{attribute 'linkalways'} 
{attribute 'no_explicit_call' := 'This FB is a CLASS and must be accessed using methods or properties'}
{attribute 'enable_dynamic_creation'}
FUNCTION_BLOCK _ETcVnDiffusivityTypeKAZE EXTENDS EnumDatatypeBase
VAR
	localData : ETcVnDiffusivityTypeKAZE;
	activeData : REFERENCE TO ETcVnDiffusivityTypeKAZE;
	enumBaseDatatype : _DINT(localData);
END_VAR

METHOD PRIVATE AddLocalEnumeration
VAR_INPUT
	Enumeration : T_MAXSTRING;
	Value : ETcVnDiffusivityTypeKAZE;
END_VAR
AddEnumeration(Enumeration, Value);
END_METHOD

PROPERTY PUBLIC Address : PVOID
GET
Address := ADR(activeData);
END_GET
END_PROPERTY

METHOD PUBLIC ClearReference
VAR_INPUT
END_VAR
activeData REF= localData;
SetBaseDatatypeReference();
END_METHOD

METHOD PUBLIC Clone : I_Datatype
VAR
    pClone : POINTER TO _ETcVnDiffusivityTypeKAZE;
END_VAR
pClone := __NEW(_ETcVnDiffusivityTypeKAZE(InitialValue := Value));
Clone := pClone^;
END_METHOD

METHOD FB_init : BOOL
VAR_INPUT
	bInitRetains : BOOL; // if TRUE, the retain variables are initialized (warm start / cold start)
	bInCopyCode : BOOL;  // if TRUE, the instance afterwards gets moved into the copy code (online change)
	InitialValue : ETcVnDiffusivityTypeKAZE;
END_VAR
localData := InitialValue;
AddBaseDatatype(enumBaseDatatype);
ClearReference();

AddLocalEnumeration('TCVN_DT1_KAZE_PM_G1', ETcVnDiffusivityTypeKAZE.TCVN_DT1_KAZE_PM_G1);
AddLocalEnumeration('TCVN_DT1_KAZE_PM_G2', ETcVnDiffusivityTypeKAZE.TCVN_DT1_KAZE_PM_G2);
AddLocalEnumeration('TCVN_DT1_KAZE_WEICKERT', ETcVnDiffusivityTypeKAZE.TCVN_DT1_KAZE_WEICKERT);
AddLocalEnumeration('TCVN_DT1_KAZE_CHARBONNIER', ETcVnDiffusivityTypeKAZE.TCVN_DT1_KAZE_CHARBONNIER);
END_METHOD

PROPERTY PUBLIC Identifier : T_MAXSTRING
GET
Identifier := 'ETcVnDiffusivityTypeKAZE';
END_GET
END_PROPERTY

METHOD IsEnumeratorValueEqual : BOOL
VAR_INPUT
	Enumerator : I_KeyValueForwardEnumerator;
END_VAR
VAR
	storedValue : ETcVnDiffusivityTypeKAZE;
END_VAR
IF NOT Enumerator.TryGet(storedValue) THEN
	RETURN;
END_IF

IsEnumeratorValueEqual := storedValue = activeData;
END_METHOD

METHOD PUBLIC MakeReferenceTo
VAR_INPUT
	ReferenceTarget : REFERENCE TO ETcVnDiffusivityTypeKAZE;
END_VAR
activeData REF= ReferenceTarget;
SetBaseDatatypeReference();
END_METHOD

METHOD PROTECTED SetBaseDatatypeReference
VAR_INPUT
END_VAR
enumBaseDatatype.MakeReferenceTo(activeData);
END_METHOD

PROPERTY PUBLIC Size : UDINT
GET
Size := SIZEOF(activeData);
END_GET
END_PROPERTY

METHOD TryMakeReferenceTo : BOOL
VAR_INPUT
	Target : I_Datatype;
END_VAR
VAR
	pTargetData : POINTER TO ETcVnDiffusivityTypeKAZE;
END_VAR
IF NOT IsEquivalentTo(Target) THEN
	RETURN;
END_IF

pTargetData := Target.Address;
activeData REF= pTargetData^;
SetBaseDatatypeReference();
TryMakeReferenceTo := TRUE;
END_METHOD

PROPERTY PUBLIC Value : ETcVnDiffusivityTypeKAZE
GET
Value := activeData;
END_GET
SET
activeData := Value;
END_SET
END_PROPERTY

END_FUNCTION_BLOCK

(* stored: Version 1.1.0.1, ProductVersion 3.1.4024.13
   POU _ETcVnDiffusivityTypeKAZE: Id {44374c61-c9bd-0cab-393d-297717105bca}, SpecialFunc None
   Folder Core: Id {507ad552-1a96-06b7-1014-67780bd79b50}
   Folder Protected: Id {5e5f0103-104f-012f-2f7a-8d2f1831477c}
   Folder Customize: Id {4ca7ae8a-f36f-0eff-168a-c4a71def487c}
   Folder Constructor: Id {4a35ecab-65c6-05f2-3990-6cd626664b1a}
   Folder Private: Id {65a0f632-1e0a-0b4e-3781-5e53d2f06e3e}
   Folder Protected: Id {3267a9e5-49f7-0333-3e46-0746b0a5155d}
   Method AddLocalEnumeration: Id {193da0fa-b225-078e-1efa-5d446f7f2019}
   Property Address: Id {75d69cb2-dc34-0528-05ab-423b868e9b21}
   Get Get: Id {0de30afa-010f-0dbe-05e8-27a9c0965c2e}
   Method ClearReference: Id {055d39ea-9ffe-0148-1d30-f94c6ea0c632}
   Method Clone: Id {e7a01f23-7495-08fd-3636-b93cedf8ea9f}
   Method FB_init: Id {b870753f-b0e0-0c96-0f16-2b9630490119}
   Property Identifier: Id {d9949398-e8f3-035c-240e-a2d0437df2b9}
   Get Get: Id {69e1f71d-a0de-0328-12ed-8735f368a6c2}
   Method IsEnumeratorValueEqual: Id {36bbac34-d46f-0c38-0478-81c0a8dab38a}
   Method MakeReferenceTo: Id {1f477ed0-ed9e-0078-0cd3-005b789e0181}
   Method SetBaseDatatypeReference: Id {b2d1e994-0bdd-05ad-2884-650b78561805}
   Property Size: Id {9d57421f-5cce-07dd-1f7e-8b9186e3e2aa}
   Get Get: Id {3a81bb60-6664-0a7d-357c-edea8b161b3f}
   Method TryMakeReferenceTo: Id {bc679ca3-2a8e-0a38-253e-b96540c54a4c}
   Property Value: Id {3fb21544-a445-01b2-04d7-57657683f049}
   Get Get: Id {fa3098d9-d771-06d1-277f-a4f2aa37df7a}
   Set Set: Id {c183e105-ed4f-0d98-317c-d3e21dcc3ca0} *)
